(* PLC project KinIn_v3.project, CODESYS CODESYS V3.5 SP19 *)
(* stored: creationDateTime 2025-01-20T16:25:15.7592113, modificationDateTime 2025-01-20T16:17:39.6822999 *)

FUNCTION_BLOCK getInvKinematics_Body
  VAR_INPUT
    M : ARRAY[1..4, 1..4] OF REAL;
    T : ARRAY[1..4, 1..4] OF REAL;
    eomg : REAL;
    ev : REAL;
    {attribute 'variable_length_array_original_scope' := 'Inout'}
    {attribute 'variable_length_array' := 'ARRAY[*,*] OF REAL'}
    {attribute 'Dimensions' := '2'}
    Blist : POINTER TO REAL;
    {attribute 'variable_length_array_original_scope' := 'Inout'}
    {attribute 'variable_length_array' := 'ARRAY[*] OF REAL'}
    {attribute 'Dimensions' := '1'}
    thetalist0 : POINTER TO REAL;
    {attribute 'variable_length_array_original_scope' := 'Inout'}
    {attribute 'variable_length_array' := 'ARRAY[*] OF REAL'}
    {attribute 'Dimensions' := '1'}
    thetalist : POINTER TO REAL;  (* as output *)
  END_VAR
  VAR_OUTPUT
    success : BOOL;
  END_VAR
  VAR
    pInv : pInv;
    BodyJacobian : BodyJacobian;
    getFwdKinematics_Body : getFwdKinematics_Body;
    fastInverseTransform : fastInverseTransform;
    MatMul : MatMul;
    Exp_se3_fromTrans : Exp_se3_fromTrans;
    se3ToSpatialVel : se3ToSpatialVel;
    norm : norm;
    i0 : DINT;
    i : DINT;
    i1 : DINT;
    j1 : DINT;
    maxiterations : DINT;
    MatMul_out : ARRAY[1..4, 1..4] OF REAL;
    Vb : ARRAY[1..6] OF REAL;  (* forgot which size maybe six? *)
    Vb1_3 : ARRAY[1..6] OF REAL;
    Vb4_6 : ARRAY[1..6] OF REAL;
    Jb : ARRAY[1..GVL.pInv_dim1, 1..GVL.pInv_dim2] OF REAL;  (* maybe in inout because of size *)
    normValue1_3 : REAL;
    normValue4_6 : REAL;
    err : BOOL;
    pInvMatrix : ARRAY[1..GVL.pInv_dim2, 1..GVL.pInv_dim1] OF REAL;
    temp_vect : ARRAY[1..GVL.nJoints] OF REAL;
  END_VAR

            i0:=1;
FOR i0:=1 TO UPPER_BOUND(thetalist,1) DO
	thetalist[i0] := thetalist0[i0];
END_FOR

i := 0;
maxiterations:= 20;

getFwdKinematics_Body(M:=M , Blist:=Blist , thetalist:=thetalist);
fastInverseTransform(T:=getFwdKinematics_Body.T);
MatMul(mat1:=fastInverseTransform.invT , mat2:=T ,
	 MatResult:=MatMul_out );
Exp_se3_fromTrans(T:= MatMul_out);
se3ToSpatialVel(se3mat:=Exp_se3_fromTrans.expmat ,
	 V=>Vb);

//error
Vb1_3[1]:=Vb[1];Vb1_3[2]:=Vb[2];Vb1_3[3]:=Vb[3];
norm(vector:= Vb1_3, normValue=> normValue1_3);
Vb4_6[1]:=Vb[4];Vb4_6[2]:=Vb[5];Vb4_6[3]:=Vb[6];
norm(vector:= Vb4_6, normValue=> normValue4_6);
err:=(normValue1_3>eomg) OR (normValue4_6>ev);

WHILE err AND i<maxiterations DO
	BodyJacobian(Blist:=Blist , thetalist:=thetalist , Jb:=Jb );
	pInv(matrix:=Jb , pInvMatrix=>pInvMatrix );

	//pinv ntheta x 6 by 6x1 
	i1:=1;j1:=1;
	FOR i1:=1 TO GVL.nJoints DO
		temp_vect[i1]:=0;
		FOR j1:=1 TO 6 DO
			temp_vect[i1]:=temp_vect[i1]+pInvMatrix[i1,j1]*Vb[j1];
		END_FOR
		thetalist[i1]:=thetalist[i1]+temp_vect[i1];
	END_FOR
	
	 //thetalist := thetalist + pinv(JacobianBody(Blist, thetalist)) * Vb;
	 
    i := i + 1;
	getFwdKinematics_Body(M:=M , Blist:=Blist , thetalist:=thetalist);	 
	fastInverseTransform(T:=getFwdKinematics_Body.T);
	MatMul(mat1:=fastInverseTransform.invT , mat2:=T ,
	MatResult:=MatMul_out );
	Exp_se3_fromTrans(T:= MatMul_out);	
	se3ToSpatialVel(se3mat:=Exp_se3_fromTrans.expmat ,
		 V=>Vb);
	//error
	Vb1_3[1]:=Vb[1];Vb1_3[2]:=Vb[2];Vb1_3[3]:=Vb[3];
	norm(vector:= Vb1_3, normValue=> normValue1_3);
	Vb4_6[1]:=Vb[4];Vb4_6[2]:=Vb[5];Vb4_6[3]:=Vb[6];
	norm(vector:= Vb4_6, normValue=> normValue4_6);
	err:=(normValue1_3>eomg) OR (normValue4_6>ev);
END_WHILE

success:=NOT(err);
          
END_FUNCTION_BLOCK
